FUNCTION F_CycleTime : UDINT // Returns current cycle time in [ms]
VAR_INPUT
END_VAR
VAR
	fbGetCurTaskIdx  : GETCURTASKINDEX;
END_VAR

fbGetCurTaskIdx();
F_CycleTime := _TaskInfo[fbGetCurTaskIdx.index].CycleTime / 10000;

END_FUNCTION

(* stored: Version 1.1.0.1
   POU F_CycleTime: Id {58c57735-4ca5-49aa-993a-6115c8444a6a}, SpecialFunc None *)
